PROGRAM MAIN
VAR
	deserializerGarbageCollector_TestSuite : DeserializerGarbageCollector_TestSuite;
	missingKeyDeserializationError_TestSuite :MissingKeyDeserializationError_TestSuite;
	invalidKeyDeserializationError_TestSuite : InvalidKeyDeserializationError_TestSuite;
	incorrectTypeDeserializationError_TestSuite : IncorrectTypeDeserializationError_TestSuite;
	incorrectKeyTypeDeserializationError_TestSuite : IncorrectKeyTypeDeserializationError_TestSuite;
	deserializationErrorFactory_TestSuite : DeserializationErrorFactory_TestSuite;
	customDeserializationFailedError_TestSuite : CustomDeserializationFailedError_TestSuite;
END_VAR

TcUnit.RUN();

END_PROGRAM

(* stored: Version 1.1.0.1, ProductVersion 3.1.4024.12
   POU MAIN: Id {79e56d3f-4a2f-4165-b00a-6e29260b0b9b}, SpecialFunc None *)
